PROGRAM PRG_AT2L0_SOLID
VAR
    bAT2L0_debug: BOOL := FALSE;
    nAT2L0_enableMode: ENUM_StageEnableMode := ENUM_StageEnableMode.DURING_MOTION;

    iIndex: INT;
    fbAT2L0_motion: ARRAY [1..19] OF FB_MotionStage;
    fbAT2L0_axes: ARRAY [1..19] OF POINTER TO DUT_MotionStage;
    fbAT2L0_ffo: ARRAY[1..19] OF FB_AttFFO;

    {attribute 'pytmc' := '
        pv: AT2L0:XTES:MMS
        expand: :%.2d:FILTER
    '}
    fbAT2L0_filters: ARRAY[1..19] OF DUT_SATT_Filter;

    {attribute 'pytmc' := '
        pv: AT2L0:XTES:TRANSMISSION
        field: DESC Overall transmission of AT2L0
    '}
    fTransmission: LREAL;

    {attribute 'pytmc' := '
        pv: AT2L0:XTES:MMS
        expand: :%.2d
    '}
    fbAT2L0_states: ARRAY[1..19] OF FB_PositionState1D_InOut;

    stOut: ST_PositionState  := (
        fPosition := 24,
        fDelta := 2,
        fVelocity := 6,
        bMoveOk := TRUE,
        bValid := TRUE);

    stIn: ST_PositionState  := (
        fPosition := 0,
        fDelta := 2,
        fVelocity := 6,
        bMoveOk := TRUE,
        bValid := TRUE);

    // For plotting voltage/current during debugging
    nM1CoilARaw AT %I*: UINT;
    nM1CoilBRaw AT %I*: UINT; // ..CoilBRaw is currently linked to EL7041 'Coil Voltage A'
    nM1CoilA: INT;
    nM1CoilB: INT;
    //nM1Current: INT;
    nM2CoilARaw AT %I*: UINT;
    nM2CoilBRaw AT %I*: UINT;
    nM2CoilA: INT;
    nM2CoilB: INT;
    //nM2Current: INT;
    nM3CoilARaw AT %I*: UINT;
    nM3CoilBRaw AT %I*: UINT;
    nM3CoilA: INT;
    nM3CoilB: INT;
    //nM3Current: INT;
    nM4CoilARaw AT %I*: UINT;
    nM4CoilBRaw AT %I*: UINT;
    nM4CoilA: INT;
    nM4CoilB: INT;
    //nM4Current: INT;
    nM5CoilARaw AT %I*: UINT;
    nM5CoilBRaw AT %I*: UINT;
    nM5CoilA: INT;
    nM5CoilB: INT;
    //nM5Current: INT;
    nM6CoilARaw AT %I*: UINT;
    nM6CoilBRaw AT %I*: UINT;
    nM6CoilA: INT;
    nM6CoilB: INT;
    //nM6Current: INT;
    nM7CoilARaw AT %I*: UINT;
    nM7CoilBRaw AT %I*: UINT;
    nM7CoilA: INT;
    nM7CoilB: INT;
    //nM7Current: INT;
    nM8CoilARaw AT %I*: UINT;
    nM8CoilBRaw AT %I*: UINT;
    nM8CoilA: INT;
    nM8CoilB: INT;
    //nM8Current: INT;
    nM9CoilARaw AT %I*: UINT;
    nM9CoilBRaw AT %I*: UINT;
    nM9CoilA: INT;
    nM9CoilB: INT;
    //nM9Current: INT;
    nM10CoilARaw AT %I*: UINT;
    nM10CoilBRaw AT %I*: UINT;
    nM10CoilA: INT;
    nM10CoilB: INT;
    //nM10Current: INT;
    nM11CoilARaw AT %I*: UINT;
    nM11CoilBRaw AT %I*: UINT;
    nM11CoilA: INT;
    nM11CoilB: INT;
    //nM11Current: INT;
    nM12CoilARaw AT %I*: UINT;
    nM12CoilBRaw AT %I*: UINT;
    nM12CoilA: INT;
    nM12CoilB: INT;
    //nM12Current: INT;
    nM13CoilARaw AT %I*: UINT;
    nM13CoilBRaw AT %I*: UINT;
    nM13CoilA: INT;
    nM13CoilB: INT;
    //nM13Current: INT;
    nM14CoilARaw AT %I*: UINT;
    nM14CoilBRaw AT %I*: UINT;
    nM14CoilA: INT;
    nM14CoilB: INT;
    //nM14Current: INT;
    nM15CoilARaw AT %I*: UINT;
    nM15CoilBRaw AT %I*: UINT;
    nM15CoilA: INT;
    nM15CoilB: INT;
    //nM15Current: INT;
    nM16CoilARaw AT %I*: UINT;
    nM16CoilBRaw AT %I*: UINT;
    nM16CoilA: INT;
    nM16CoilB: INT;
    //nM16Current: INT;
    nM17CoilARaw AT %I*: UINT;
    nM17CoilBRaw AT %I*: UINT;
    nM17CoilA: INT;
    nM17CoilB: INT;
    //nM17Current: INT;
    nM18CoilARaw AT %I*: UINT;
    nM18CoilBRaw AT %I*: UINT;
    nM18CoilA: INT;
    nM18CoilB: INT;
    //nM18Current: INT;
    nM19CoilARaw AT %I*: UINT;
    nM19CoilBRaw AT %I*: UINT;
    nM19CoilA: INT;
    nM19CoilB: INT;
    //nM19Current: INT;

    stFilter : REFERENCE TO DUT_SATT_Filter;
    fFilterDensity : LREAL;
    fFilterAtomicMass : LREAL;
    fbAtomicMass : FB_AtomicMass;
    fbAttenuatorElementDensity : FB_AttenuatorElementDensity;
    fAbsorptionConstant : LREAL;
    bError : BOOL;

END_VAR


fbAT2L0_axes[1]:= ADR(Main.M1);
fbAT2L0_axes[2]:= ADR(Main.M2);
fbAT2L0_axes[3]:= ADR(Main.M3);
fbAT2L0_axes[4]:= ADR(Main.M4);
fbAT2L0_axes[5]:= ADR(Main.M5);
fbAT2L0_axes[6]:= ADR(Main.M6);
fbAT2L0_axes[7]:= ADR(Main.M7);
fbAT2L0_axes[8]:= ADR(Main.M8);
fbAT2L0_axes[9]:= ADR(Main.M9);
fbAT2L0_axes[10]:= ADR(Main.M10);
fbAT2L0_axes[11]:= ADR(Main.M11);
fbAT2L0_axes[12]:= ADR(Main.M12);
fbAT2L0_axes[13]:= ADR(Main.M13);
fbAT2L0_axes[14]:= ADR(Main.M14);
fbAT2L0_axes[15]:= ADR(Main.M15);
fbAT2L0_axes[16]:= ADR(Main.M16);
fbAT2L0_axes[17]:= ADR(Main.M17);
fbAT2L0_axes[18]:= ADR(Main.M18);
fbAT2L0_axes[19]:= ADR(Main.M19);

(* Not a filter *)
fbAT2L0_filters[ 1].fFilterThickness_um := 0;
fbAT2L0_filters[ 1].sFilterMaterial     := '';

fbAT2L0_filters[ 2].fFilterThickness_um := 1280.0;
fbAT2L0_filters[ 2].sFilterMaterial     := 'C';
fbAT2L0_filters[ 3].fFilterThickness_um := 320.0;
fbAT2L0_filters[ 3].sFilterMaterial     := 'C';
fbAT2L0_filters[ 4].fFilterThickness_um := 640.0;
fbAT2L0_filters[ 4].sFilterMaterial     := 'C';
fbAT2L0_filters[ 5].fFilterThickness_um := 160.0;
fbAT2L0_filters[ 5].sFilterMaterial     := 'C';
fbAT2L0_filters[ 6].fFilterThickness_um := 80.0;
fbAT2L0_filters[ 6].sFilterMaterial     := 'C';
fbAT2L0_filters[ 7].fFilterThickness_um := 40.0;
fbAT2L0_filters[ 7].sFilterMaterial     := 'C';
fbAT2L0_filters[ 8].fFilterThickness_um := 20.0;
fbAT2L0_filters[ 8].sFilterMaterial     := 'C';
fbAT2L0_filters[ 9].fFilterThickness_um := 10.0;
fbAT2L0_filters[ 9].sFilterMaterial     := 'C';

fbAT2L0_filters[10].fFilterThickness_um := 10240.0;
fbAT2L0_filters[10].sFilterMaterial     := 'Si';
fbAT2L0_filters[11].fFilterThickness_um := 5120.0;
fbAT2L0_filters[11].sFilterMaterial     := 'Si';
fbAT2L0_filters[12].fFilterThickness_um := 2560.0;
fbAT2L0_filters[12].sFilterMaterial     := 'Si';
fbAT2L0_filters[13].fFilterThickness_um := 1280.0;
fbAT2L0_filters[13].sFilterMaterial     := 'Si';
fbAT2L0_filters[14].fFilterThickness_um := 640.0;
fbAT2L0_filters[14].sFilterMaterial     := 'Si';
fbAT2L0_filters[15].fFilterThickness_um := 320.0;
fbAT2L0_filters[15].sFilterMaterial     := 'Si';
fbAT2L0_filters[16].fFilterThickness_um := 160.0;
fbAT2L0_filters[16].sFilterMaterial     := 'Si';
fbAT2L0_filters[17].fFilterThickness_um := 80.0;
fbAT2L0_filters[17].sFilterMaterial     := 'Si';
fbAT2L0_filters[18].fFilterThickness_um := 40.0;
fbAT2L0_filters[18].sFilterMaterial     := 'Si';
fbAT2L0_filters[19].fFilterThickness_um := 20.0;
fbAT2L0_filters[19].sFilterMaterial     := 'Si';

IF bAT2L0_debug THEN
    nAT2L0_enableMode := ENUM_StageEnableMode.ALWAYS;
ELSE
    nAT2L0_enableMode := ENUM_StageEnableMode.DURING_MOTION;
END_IF


(* Recalculate the overall transmission below *)
fTransmission := 1.0;

FOR iIndex := 1 TO 19 DO
    fbAT2L0_motion[iIndex](stMotionStage := fbAT2L0_axes[iIndex]^);
    fbAT2L0_axes[iIndex]^.nEnableMode := nAT2L0_enableMode;
    fbAT2L0_axes[iIndex]^.bHardwareEnable := TRUE;
    fbAT2L0_axes[iIndex]^.bPowerSelf := TRUE;
    stFilter REF= fbAT2L0_filters[iIndex];

    fbAT2L0_states[iIndex](
        stMotionStage := fbAT2L0_axes[iIndex]^,
        stOut := stOut,
        stIn := stIn);

    fbAT2L0_ffo[iIndex](
        stMotionStage := fbAT2L0_axes[iIndex]^,
        enumState := fbAT2L0_states[iIndex].eStateGet,
        fbFFHWO := GVL.fbFastFaultOutput1);

    IF fbAT2L0_states[iIndex].eStateGet = ENUM_EpicsInOut.UNKNOWN THEN
        stFilter.fTransmission := 0.0;
    ELSIF fbAT2L0_states[iIndex].eStateGet = ENUM_EpicsInOut.OUT OR stFilter.sFilterMaterial = '' THEN
        stFilter.fTransmission := 1.0;
    ELSE
        fbAtomicMass(sName:=stFilter.sFilterMaterial, fValue=>fFilterAtomicMass);
        fbAttenuatorElementDensity(sName:=stFilter.sFilterMaterial, fDensity=>fFilterDensity);

        fAbsorptionConstant := F_CalculateAbsorptionConstant(
            sElement:=stFilter.sFilterMaterial,
            fEnergyEV:=PMPS_GVL.stCurrentBeamParameters.neV,
            fDensity_gm3:=fFilterDensity,
            fAtomicWeight:=fFilterAtomicMass,
            bError=>bError,
        );
        stFilter.fTransmission := F_CalculateTransmission(
            fAbsorptionConstant:=fAbsorptionConstant,
            fThickness_in_m:=stFilter.fFilterThickness_um * 1.0E-6
        );
    END_IF

    fTransmission := fTransmission * stFilter.fTransmission;
END_FOR

IF fbAT2L0_states[1].eStateGet = ENUM_EpicsInOut.IN THEN
    (* Inspection mirror blocks the beam *)
    GVL.rCurTrans[PMPS.L_Attenuators.AT2L0].nTran := 0.0;
    (* TODO fast fault as well *)
ELSE
    GVL.rCurTrans[PMPS.L_Attenuators.AT2L0].nTran := LREAL_TO_REAL(fTransmission);
END_IF

iIndex := 0;

nM1CoilA := UINT_TO_INT(nM1CoilARaw);
nM1CoilB := UINT_TO_INT(nM1CoilBRaw);
//nM1Current := ABS(nM1CoilA) + ABS(nM1CoilB);
nM2CoilA := UINT_TO_INT(nM2CoilARaw);
nM2CoilB := UINT_TO_INT(nM2CoilBRaw);
//nM2Current := ABS(nM2CoilA) + ABS(nM2CoilB);
nM3CoilA := UINT_TO_INT(nM3CoilARaw);
nM3CoilB := UINT_TO_INT(nM3CoilBRaw);
//nM3Current := ABS(nM3CoilA) + ABS(nM3CoilB);
nM4CoilA := UINT_TO_INT(nM4CoilARaw);
nM4CoilB := UINT_TO_INT(nM4CoilBRaw);
//nM4Current := ABS(nM4CoilA) + ABS(nM4CoilB);
nM5CoilA := UINT_TO_INT(nM5CoilARaw);
nM5CoilB := UINT_TO_INT(nM5CoilBRaw);
//nM5Current := ABS(nM5CoilA) + ABS(nM5CoilB);
nM5CoilA := UINT_TO_INT(nM5CoilARaw);
nM5CoilB := UINT_TO_INT(nM5CoilBRaw);
//nM5Current := ABS(nM5CoilA) + ABS(nM5CoilB);
nM6CoilA := UINT_TO_INT(nM6CoilARaw);
nM6CoilB := UINT_TO_INT(nM6CoilBRaw);
//nM6Current := ABS(nM6CoilA) + ABS(nM6CoilB);
nM7CoilA := UINT_TO_INT(nM7CoilARaw);
nM7CoilB := UINT_TO_INT(nM7CoilBRaw);
//nM7Current := ABS(nM7CoilA) + ABS(nM7CoilB);
nM8CoilA := UINT_TO_INT(nM8CoilARaw);
nM8CoilB := UINT_TO_INT(nM8CoilBRaw);
//nM8Current := ABS(nM9CoilA) + ABS(nM9CoilB);
nM9CoilA := UINT_TO_INT(nM9CoilARaw);
nM9CoilB := UINT_TO_INT(nM9CoilBRaw);
//nM9Current := ABS(nM9CoilA) + ABS(nM9CoilB);
nM10CoilA := UINT_TO_INT(nM10CoilARaw);
nM10CoilB := UINT_TO_INT(nM10CoilBRaw);
//nM10Current := ABS(nM10CoilA) + ABS(nM10CoilB);
nM11CoilA := UINT_TO_INT(nM11CoilARaw);
nM11CoilB := UINT_TO_INT(nM11CoilBRaw);
//nM11Current := ABS(nM11CoilA) + ABS(nM11CoilB);
nM12CoilA := UINT_TO_INT(nM12CoilARaw);
nM12CoilB := UINT_TO_INT(nM12CoilBRaw);
//nM12Current := ABS(nM12CoilA) + ABS(nM12CoilB);
nM13CoilA := UINT_TO_INT(nM13CoilARaw);
nM13CoilB := UINT_TO_INT(nM13CoilBRaw);
//nM13Current := ABS(nM13CoilA) + ABS(nM13CoilB);
nM14CoilA := UINT_TO_INT(nM14CoilARaw);
nM14CoilB := UINT_TO_INT(nM14CoilBRaw);
//nM14Current := ABS(nM14CoilA) + ABS(nM14CoilB);
nM15CoilA := UINT_TO_INT(nM15CoilARaw);
nM15CoilB := UINT_TO_INT(nM15CoilBRaw);
//nM15Current := ABS(nM15CoilA) + ABS(nM15CoilB);
nM16CoilA := UINT_TO_INT(nM16CoilARaw);
nM16CoilB := UINT_TO_INT(nM16CoilBRaw);
//nM16Current := ABS(nM16CoilA) + ABS(nM16CoilB);
nM17CoilA := UINT_TO_INT(nM17CoilARaw);
nM17CoilB := UINT_TO_INT(nM17CoilBRaw);
//nM17Current := ABS(nM17CoilA) + ABS(nM17CoilB);
nM18CoilA := UINT_TO_INT(nM18CoilARaw);
nM18CoilB := UINT_TO_INT(nM18CoilBRaw);
//nM18Current := ABS(nM2CoilA) + ABS(nM18CoilB);
nM19CoilA := UINT_TO_INT(nM19CoilARaw);
nM19CoilB := UINT_TO_INT(nM19CoilBRaw);
//nM19Current := ABS(nM2CoilA) + ABS(nM2CoilB);

END_PROGRAM

(* stored: Version 1.1.0.1
   POU PRG_AT2L0_SOLID: Id {6180f524-6468-4c61-b137-11e8cfa13685}, SpecialFunc None *)
